FUNCTION "LGF_SplitDWordToBytes" : Void
TITLE = LGF_SplitDWordToBytes
{ S7_Optimized_Access := 'TRUE' }
AUTHOR : Siemens_Digital_Industry
FAMILY : LGF
NAME : LGF_SplitDWordToBytes
//This function splits a DWord variable into 4 Byte variables.
   VAR_INPUT
      doubleWord : DWord;   // Bit sequence to be split
   END_VAR

   VAR_OUTPUT
      byte3 : Byte;   // Output Byte 3 - MSB
      byte2 : Byte;   // Output Byte 2
      byte1 : Byte;   // Output Byte 1
      byte0 : Byte;   // Output Byte 0 - LSB
   END_VAR


BEGIN
	REGION BLOCK INFO HEADER
	  //===============================================================================
	  // SIEMENS AG / (c)Copyright 2018
	  //-------------------------------------------------------------------------------
	  // Title:            LGF_SplitDWordToBytes
	  // Comment/Function: This function splits a DWord variable into 4 Byte variables.
	  // Library/Family:   LGF (Library General Functions)
	  // Author:           Siemens Digital Industry Support
	  // Tested with:      S7-PLCSIM Advanced V2.0 SP1
	  // Engineering:      TIA Portal V14 / V14SP1
	  // Restrictions:     ENO disabled - no error handling, no failure possible.
	  // Requirements:     PLC (S7-1200 / S7-1500)
	  //-------------------------------------------------------------------------------
	  // Change log table:
	  // Version  | Date       | Expert in charge       | Changes applied
	  //----------|------------|------------------------|------------------------------
	  // 01.00.00 | 20.06.2019 | Simatic Systems Support
	  //                         First release
	  // 03.00.00 | 23.04.2020 | Simatic Systems Support | Set version to V3.0.0
	  //                         harmonize the version of the whole library
	  // 03.00.01 | 22.02.2021 | Simatic Systems Support
	  //                         Insert documentation
	  //=============================================================================
	END_REGION

	REGION OUTPUT
	  // get the bytes by slice access
	  #byte3 := #doubleWord.%B3;
	  #byte2 := #doubleWord.%B2;
	  #byte1 := #doubleWord.%B1;
	  #byte0 := #doubleWord.%B0;
	  // no error handling needed
	  ENO := TRUE;
	END_REGION

END_FUNCTION

